// TIA Portal V20 export
FUNCTION_BLOCK "SysLinMotC1150"   // FB2080, FBD
TITLE = manage the positioning over the "extended bus positioning" [6Word]
{ S7_Optimized_Access := 'TRUE' }
AUTHOR : MiCROTEC
VERSION : 1.6
// -2019.12 : Martin
// stored: AutoNumber false, MemoryReserve 100, SetENOAutomatically false
   VAR_INPUT
      adr { ExternalAccessible := 'False'; ExternalVisible := 'False'; ExternalWritable := 'False'} : HW_IO;   // I/O address
      adrMc1 { ExternalAccessible := 'False'; ExternalVisible := 'False'; ExternalWritable := 'False'} : HW_IO;   // I/O address monitoring channel 1
      adrMc2 { ExternalAccessible := 'False'; ExternalVisible := 'False'; ExternalWritable := 'False'} : HW_IO;   // I/O address monitoring channel 2
      area { ExternalAccessible := 'False'; ExternalVisible := 'False'; ExternalWritable := 'False'} : Bool;   // 1=Safety area on
      areaDel { ExternalAccessible := 'False'; ExternalVisible := 'False'; ExternalWritable := 'False'} : Bool;   // 1=safety area on off-delayed
      auto { ExternalAccessible := 'False'; ExternalVisible := 'False'; ExternalWritable := 'False'} : Bool;   // automatic
      manP { ExternalAccessible := 'False'; ExternalVisible := 'False'; ExternalWritable := 'False'} : Bool;   // manual plus
      manM { ExternalAccessible := 'False'; ExternalVisible := 'False'; ExternalWritable := 'False'} : Bool;   // manual minus
      enable { ExternalAccessible := 'False'; ExternalVisible := 'False'; ExternalWritable := 'False'} : Bool;   // enable positioning
      enableP { ExternalAccessible := 'False'; ExternalVisible := 'False'; ExternalWritable := 'False'} : Bool;   // release plus
      enableM { ExternalAccessible := 'False'; ExternalVisible := 'False'; ExternalWritable := 'False'} : Bool;   // release minus
      ref { ExternalAccessible := 'False'; ExternalVisible := 'False'; ExternalWritable := 'False'} : Bool;   // reference
      ack { ExternalAccessible := 'False'; ExternalVisible := 'False'; ExternalWritable := 'False'} : Bool;   // fault acknowledge
      lampTest { ExternalAccessible := 'False'; ExternalVisible := 'False'; ExternalWritable := 'False'} : Bool;   // lamptest
      PwrSupMot { ExternalAccessible := 'False'; ExternalVisible := 'False'; ExternalWritable := 'False'} : Bool;   // 1=power supply motor ok / 1=motor protection switch ok
      PwrSupCtrl { ExternalAccessible := 'False'; ExternalVisible := 'False'; ExternalWritable := 'False'} : Bool;   // 1=power supply controller ok / 1=Motor protection switch brake ok
      tolerance { ExternalAccessible := 'False'; ExternalVisible := 'False'; ExternalWritable := 'False'} : Real;   // tolerance for output signal position ok
      mode { ExternalAccessible := 'False'; ExternalVisible := 'False'; ExternalWritable := 'False'} : Int;   // 1=VAI / 2=SIN VA / 3=Bestehorn VAJ
      target { ExternalAccessible := 'False'; ExternalVisible := 'False'; ExternalWritable := 'False'} : Real;   // target position [mm] / target position
      speed { ExternalAccessible := 'False'; ExternalVisible := 'False'; ExternalWritable := 'False'} : Real;   // target speed [m/s ] / target speed [ 1/min ]
      Acc { ExternalAccessible := 'False'; ExternalVisible := 'False'; ExternalWritable := 'False'} : Real;   // acceleration [m/s2] / start ramp [ms]
      Dec { ExternalAccessible := 'False'; ExternalVisible := 'False'; ExternalWritable := 'False'} : Real;   // deceleration [m/s2] / stop ramp [ms]
      jerk { ExternalAccessible := 'False'; ExternalVisible := 'False'; ExternalWritable := 'False'} : Real;   // jerk [m/s3]
   END_VAR
   VAR_OUTPUT
      comOk { ExternalAccessible := 'False'; ExternalVisible := 'False'; ExternalWritable := 'False'} : Bool;   // frequency converter communication ok
      ready { ExternalAccessible := 'False'; ExternalVisible := 'False'; ExternalWritable := 'False'} : Bool;   // frequency converter ready
      encAct { ExternalAccessible := 'False'; ExternalVisible := 'False'; ExternalWritable := 'False'} : DInt;   // actual position [inc]
      actual { ExternalAccessible := 'False'; ExternalVisible := 'False'; ExternalWritable := 'False'} : Real;   // actual position
      refOk { ExternalAccessible := 'False'; ExternalVisible := 'False'; ExternalWritable := 'False'} : Bool;   // reference ok
      refRun { ExternalAccessible := 'False'; ExternalVisible := 'False'; ExternalWritable := 'False'} : Bool;   // reference run active
      posOk { ExternalAccessible := 'False'; ExternalVisible := 'False'; ExternalWritable := 'False'} : Bool;   // position ok
      lamp { ExternalAccessible := 'False'; ExternalVisible := 'False'; ExternalWritable := 'False'} : Bool;   // indication lamp
      err { ExternalAccessible := 'False'; ExternalVisible := 'False'; ExternalWritable := 'False'} : Bool;   // fault
      errEnc { ExternalAccessible := 'False'; ExternalVisible := 'False'; ExternalWritable := 'False'} : Bool;   // fault encoder
      war { ExternalAccessible := 'False'; ExternalVisible := 'False'; ExternalWritable := 'False'} : Bool;   // warning
   END_VAR
   VAR_IN_OUT
      Mot : "TypeMotor";   // data motor
   END_VAR
   VAR
      var { ExternalAccessible := 'False'; ExternalVisible := 'False'; ExternalWritable := 'False'} : Struct
         "bool" : Bool;
         "byte" : Byte;
         "word" : Word;
         "dword" : DWord;
         "int" : Int;
         "dint" : DInt;
         "real" : Real;
         s5time : S5Time;
         "time" : Time;
         hm : Array[1..16] of Bool;
         fm : Array[1..16] of Bool;
      END_STRUCT;
      Rd { ExternalAccessible := 'False'; ExternalVisible := 'False'; ExternalWritable := 'False'} : "TypeLinmotRd";
      RdMc1 { ExternalAccessible := 'False'; ExternalVisible := 'False'; ExternalWritable := 'False'} : DInt;   // actual velocity
      RdMc2 { ExternalAccessible := 'False'; ExternalVisible := 'False'; ExternalWritable := 'False'} : DInt;   // actual error code
      Sd { ExternalAccessible := 'False'; ExternalVisible := 'False'; ExternalWritable := 'False'} : "TypeLinmotSd";
      T { ExternalAccessible := 'False'; ExternalVisible := 'False'; ExternalWritable := 'False'} : Array[1..8] of IEC_TIMER;
      errNrOld { ExternalAccessible := 'False'; ExternalVisible := 'False'; ExternalWritable := 'False'} : UDInt;
      man { ExternalAccessible := 'False'; ExternalVisible := 'False'; ExternalWritable := 'False'} : Bool;
      autoOld { ExternalAccessible := 'False'; ExternalVisible := 'False'; ExternalWritable := 'False'} : Bool;
      errGen { ExternalAccessible := 'False'; ExternalVisible := 'False'; ExternalWritable := 'False'} : Bool;
      enOnDel { ExternalAccessible := 'False'; ExternalVisible := 'False'; ExternalWritable := 'False'} : Bool;
      MotEnable { ExternalAccessible := 'False'; ExternalVisible := 'False'; ExternalWritable := 'False'} : Bool;
      MotSwitchOn { ExternalAccessible := 'False'; ExternalVisible := 'False'; ExternalWritable := 'False'} : Bool;
      statReady { ExternalAccessible := 'False'; ExternalVisible := 'False'; ExternalWritable := 'False'} : Bool;
      statCtrlAuto { ExternalAccessible := 'False'; ExternalVisible := 'False'; ExternalWritable := 'False'} : Bool;
      TarPos { ExternalAccessible := 'False'; ExternalVisible := 'False'; ExternalWritable := 'False'} : Real;
      TarCurrent { ExternalAccessible := 'False'; ExternalVisible := 'False'; ExternalWritable := 'False'} : Real;
      TimeResetHome { ExternalAccessible := 'False'; ExternalVisible := 'False'; ExternalWritable := 'False'} : TON_TIME;
      targetOld { ExternalAccessible := 'False'; ExternalVisible := 'False'; ExternalWritable := 'False'} : Real;
      StartPos { ExternalAccessible := 'False'; ExternalVisible := 'False'; ExternalWritable := 'False'} : Bool;
      PosTolOk { ExternalAccessible := 'False'; ExternalVisible := 'False'; ExternalWritable := 'False'} : Bool;
      TimeStartPos { ExternalAccessible := 'False'; ExternalVisible := 'False'; ExternalWritable := 'False'} : TP_TIME;
      McPar4 { ExternalAccessible := 'False'; ExternalVisible := 'False'; ExternalWritable := 'False'} : Real;
      Mc1 { ExternalAccessible := 'False'; ExternalVisible := 'False'; ExternalWritable := 'False'} : DInt;
      Mc2 { ExternalAccessible := 'False'; ExternalVisible := 'False'; ExternalWritable := 'False'} : DInt;
   END_VAR
   VAR_TEMP
      tempSdRetVal : Int;
      tempRdRetVal1 : Int;
      tempRdRetVal2 : Int;
      tempRdRetVal3 : Int;
      tempName : WString[20];
      tempDescription : WString[60];
      label : WString[26];
      tempString : WString;
      tempStrgPointer : Int;
      tempAck : Bool;
      tempStat : Bool;
      tempWar : Bool;
      tempOp : DInt;
      tempRd : Array[0..3] of Byte;
      tempDint : DInt;
      tempSd : Array[0..3] of Byte;
   END_VAR
   VAR_TEMP   // added for the SCL form of the ladder/FBD networks
      _w1 : Bool;
      _w2 : Bool;
   END_VAR
BEGIN

REGION Network 1 (SCL): description
   // Linmot  PL01-20x800/740-HP  Motor Stange Noale
   // control of a linmot motor
   // controller:  Linmot C1150-PN-XC-1S
   // stator:      Linmot PS01-37Sx120F-HP-N-AGI
   // stroke:      Linmot PL01-20x360/300-HP
   // creator:     Alexander Kiebacher
   // version:     1.0
   //
END_REGION

REGION Network 2: exit
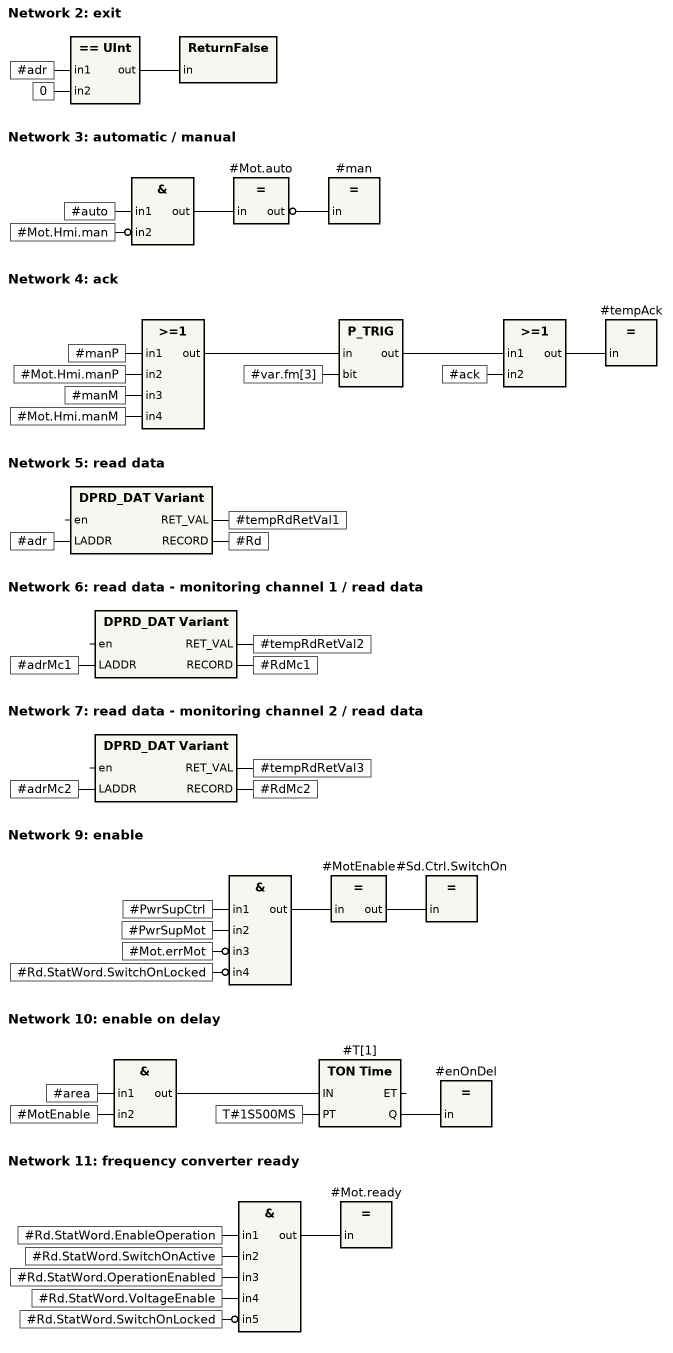
   IF #adr = 0 THEN
       ENO := FALSE;
       RETURN;
   END_IF;
END_REGION

REGION Network 3: automatic / manual
   #_w1 := #auto AND NOT #Mot.Hmi.man;
   #Mot.auto := #_w1;
   #man := NOT #_w1;
END_REGION

REGION Network 4: ack
   #_w1 := #manP OR #Mot.Hmi.manP OR #manM OR #Mot.Hmi.manM;
   #_w2 := #_w1 AND NOT #var.fm[3];   // rising edge
   #var.fm[3] := #_w1;
   #tempAck := #_w2 OR #ack;
END_REGION

REGION Network 5: read data
   #tempRdRetVal1 := DPRD_DAT(LADDR := #adr, RECORD => #Rd);
END_REGION

REGION Network 6: read data - monitoring channel 1 / read data
   #tempRdRetVal2 := DPRD_DAT(LADDR := #adrMc1, RECORD => #RdMc1);
END_REGION

REGION Network 7: read data - monitoring channel 2 / read data
   #tempRdRetVal3 := DPRD_DAT(LADDR := #adrMc2, RECORD => #RdMc2);
END_REGION

REGION Network 8 (SCL): read

   // actual position
   #tempRd[0] := #Rd.Actpos.%B0;
   #tempRd[1] := #Rd.Actpos.%B1;
   #tempRd[2] := #Rd.Actpos.%B2;
   #tempRd[3] := #Rd.Actpos.%B3;

   #Rd.Actpos.%B0 := #tempRd[3];
   #Rd.Actpos.%B1 := #tempRd[2];
   #Rd.Actpos.%B2 := #tempRd[1];
   #Rd.Actpos.%B3 := #tempRd[0];

   #encAct := #Rd.Actpos;
   #actual := DINT_TO_REAL(#Rd.Actpos) / 10000.0;

   // target position
   #tempRd[0] := #Rd.Tarpos.%B0;
   #tempRd[1] := #Rd.Tarpos.%B1;
   #tempRd[2] := #Rd.Tarpos.%B2;
   #tempRd[3] := #Rd.Tarpos.%B3;

   #Rd.Tarpos.%B0 := #tempRd[3];
   #Rd.Tarpos.%B1 := #tempRd[2];
   #Rd.Tarpos.%B2 := #tempRd[1];
   #Rd.Tarpos.%B3 := #tempRd[0];

   #TarPos := DINT_TO_REAL(#Rd.Tarpos) / 10000.0;

   // target current
   #tempRd[0] := #Rd.TarCurrent.%B0;
   #tempRd[1] := #Rd.TarCurrent.%B1;
   #tempRd[2] := #Rd.TarCurrent.%B2;
   #tempRd[3] := #Rd.TarCurrent.%B3;

   #Rd.TarCurrent.%B0 := #tempRd[3];
   #Rd.TarCurrent.%B1 := #tempRd[2];
   #Rd.TarCurrent.%B2 := #tempRd[1];
   #Rd.TarCurrent.%B3 := #tempRd[0];

   #TarCurrent := DINT_TO_REAL(#Rd.TarCurrent) / 1000.0;

   // monitoring channel 1 - target velocity [1000*m/s]
   #tempRd[0] := #RdMc1.%B0;
   #tempRd[1] := #RdMc1.%B1;
   #tempRd[2] := #RdMc1.%B2;
   #tempRd[3] := #RdMc1.%B3;

   #RdMc1.%B0 := #tempRd[3];
   #RdMc1.%B1 := #tempRd[2];
   #RdMc1.%B2 := #tempRd[1];
   #RdMc1.%B3 := #tempRd[0];

   #Mc1 := #RdMc1;

   IF #Rd.StatWord.MotionActive THEN
       IF #Mc1 >= 100 THEN
           #Mot.speedAct := DINT_TO_INT(#Mc1/1000);
       ELSIF #Mc1 <= -100 THEN
           #Mot.speedAct := DINT_TO_INT(#Mc1/1000);
       END_IF;
   ELSE
       #Mot.speedAct := 0;
   END_IF;

   // monitoring channel 2 - actual error code
   #tempRd[0] := #RdMc2.%B0;
   #tempRd[1] := #RdMc2.%B1;
   #tempRd[2] := #RdMc2.%B2;
   #tempRd[3] := #RdMc2.%B3;

   #RdMc2.%B0 := #tempRd[3];
   #RdMc2.%B1 := #tempRd[2];
   #RdMc2.%B2 := #tempRd[1];
   #RdMc2.%B3 := #tempRd[0];

   #Mc2 := #RdMc2;
END_REGION

REGION Network 9: enable
   #MotEnable := #PwrSupCtrl AND #PwrSupMot AND NOT #Mot.errMot AND NOT #Rd.StatWord.SwitchOnLocked;
   #Sd.Ctrl.SwitchOn := #MotEnable;
END_REGION

REGION Network 10: enable on delay
   #T[1].TON(IN := #area AND #MotEnable, PT := T#1S500MS);
   #enOnDel := #T[1].Q;
END_REGION

REGION Network 11: frequency converter ready
   #Mot.ready := #Rd.StatWord.EnableOperation AND #Rd.StatWord.SwitchOnActive AND #Rd.StatWord.OperationEnabled AND #Rd.StatWord.VoltageEnable AND NOT #Rd.StatWord.SwitchOnLocked;
END_REGION

REGION Network 12: ready
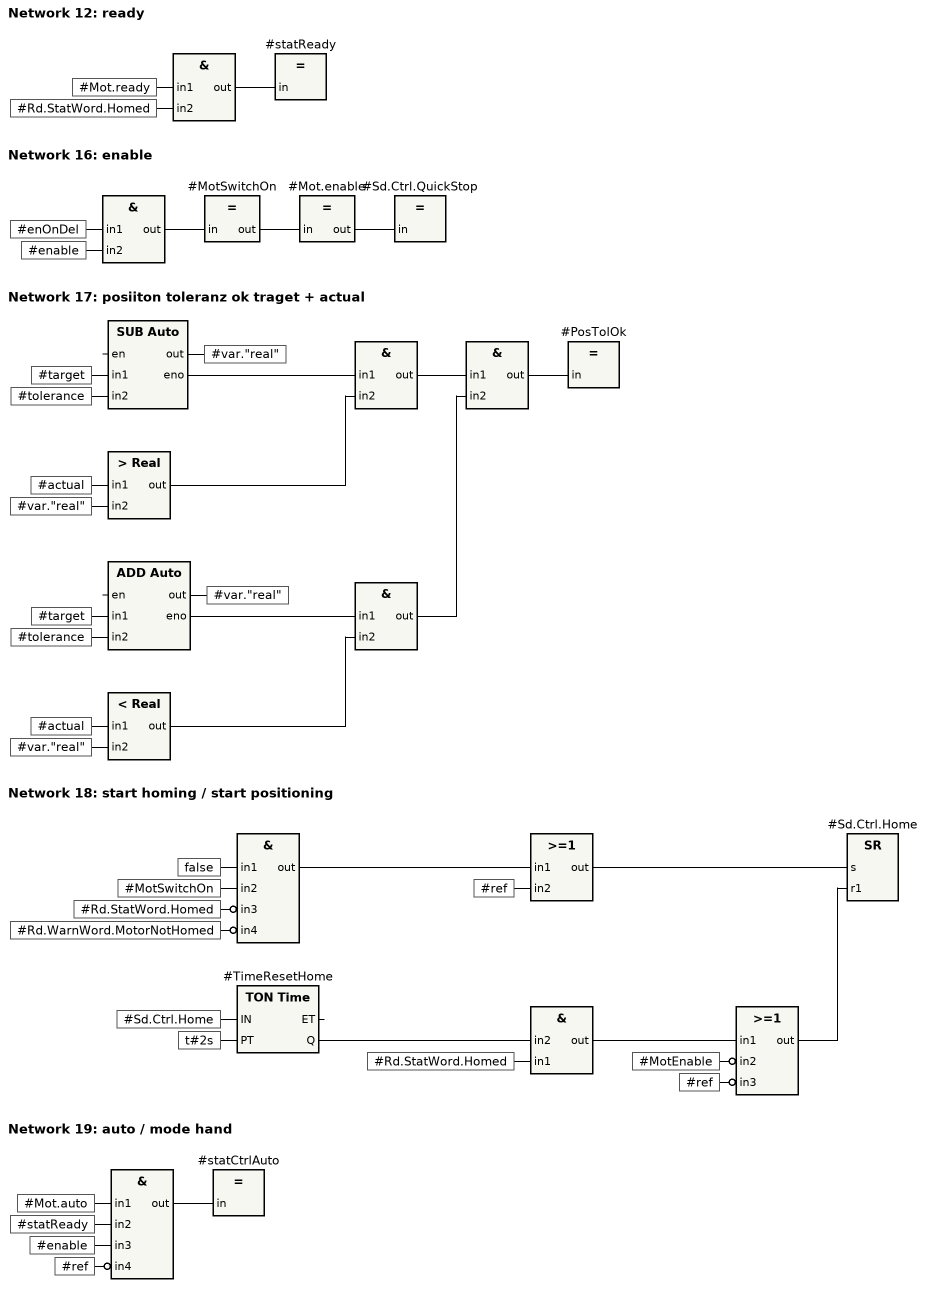
   #statReady := #Mot.ready AND #Rd.StatWord.Homed;
END_REGION

NETWORK
TITLE = test status var

      L     #Rd.StatVar.MainState;  // Op. Main State
      L     #Rd.StatVar.SubState;  // Op. Sub State

      T     #tempOp;


NETWORK
TITLE = test status word

// not used
      O     #Rd.StatWord.EventHandlerActive;
      O     #Rd.StatWord.SpecialMotionActive;
      O     #Rd.StatWord.MotionActive;
      O     #Rd.StatWord.RangeIndicator1;
      O     #Rd.StatWord.RangeIndicator2;
      =     #tempStat;


NETWORK
TITLE = test warning word

// not used
      O     #Rd.StatWord.Warning;
      O     #Rd.WarnWord.MotorHotSensor;
      O     #Rd.WarnWord.MotorShortTimerOverload;
      O     #Rd.WarnWord.MotorSupplyVoltageLow;
      O     #Rd.WarnWord.MotorSupplyVoltageHigh;
      O     #Rd.WarnWord.PositionLagAlways;
      O     #Rd.WarnWord.Res5;
      O     #Rd.WarnWord.DriveHot;
      O     #Rd.WarnWord.PTC_Sensor1Hot;
      O     #Rd.WarnWord.PTC_Sensor2Hot;
      O     #Rd.WarnWord.Res10;
      O     #Rd.WarnWord.Res11;
      O     #Rd.WarnWord.Res12;
      O     #Rd.WarnWord.Res13;
      O     #Rd.WarnWord.InterfaceWarnFlag;
      O     #Rd.WarnWord.ApplicationWarnFlag;
      =     #tempWar;


REGION Network 16: enable
   #MotSwitchOn := #enOnDel AND #enable;
   #Mot.enable := #MotSwitchOn;
   #Sd.Ctrl.QuickStop := #MotSwitchOn;
END_REGION

REGION Network 17: posiiton toleranz ok traget + actual
   #var."real" := #target - #tolerance;
   #_w1 := #actual > #var."real";
   #var."real" := #target + #tolerance;
   #PosTolOk := #_w1 AND (#actual < #var."real");
END_REGION

REGION Network 18: start homing / start positioning
   // auto reference?
   #TimeResetHome(IN := #Sd.Ctrl.Home, PT := t#2s);   // TON
   IF (false AND #MotSwitchOn AND NOT #Rd.StatWord.Homed AND NOT #Rd.WarnWord.MotorNotHomed) OR #ref THEN
       #Sd.Ctrl.Home := TRUE;   // SR flip-flop
   END_IF;
   IF (#TimeResetHome.Q AND #Rd.StatWord.Homed) OR NOT #MotEnable OR NOT #ref THEN
       #Sd.Ctrl.Home := FALSE;
   END_IF;
END_REGION

REGION Network 19: auto / mode hand
   #statCtrlAuto := #Mot.auto AND #statReady AND #enable AND NOT #ref;
END_REGION

REGION Network 20: start positioning
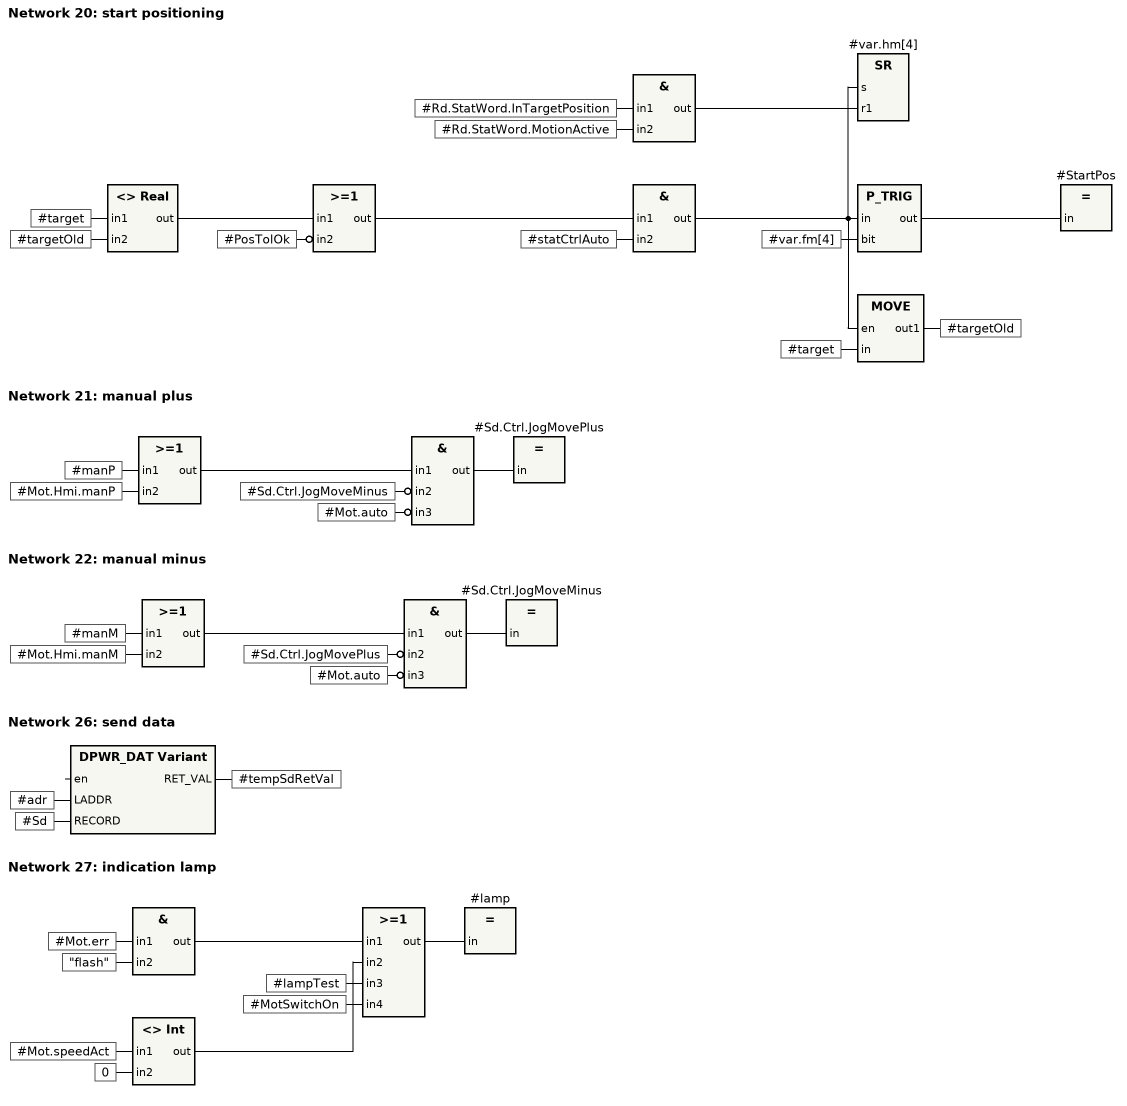
   #_w1 := ((#target <> #targetOld) OR NOT #PosTolOk) AND #statCtrlAuto;
   IF #_w1 THEN
       #var.hm[4] := TRUE;   // SR flip-flop
   END_IF;
   IF #Rd.StatWord.InTargetPosition AND #Rd.StatWord.MotionActive THEN #var.hm[4] := FALSE; END_IF;
   #_w2 := #_w1 AND NOT #var.fm[4];   // rising edge
   #var.fm[4] := #_w1;
   #StartPos := #_w2;
   IF #_w1 THEN #targetOld := #target; END_IF;
END_REGION

REGION Network 21: manual plus
   #Sd.Ctrl.JogMovePlus := (#manP OR #Mot.Hmi.manP) AND NOT #Sd.Ctrl.JogMoveMinus AND NOT #Mot.auto;
END_REGION

REGION Network 22: manual minus
   #Sd.Ctrl.JogMoveMinus := (#manM OR #Mot.Hmi.manM) AND NOT #Sd.Ctrl.JogMovePlus AND NOT #Mot.auto;
END_REGION

REGION Network 23 (SCL)

   #Sd.Ctrl.EnableOperation := TRUE;          // Forced
   #Sd.Ctrl.Abort := TRUE;                    // Forced
   #Sd.Ctrl.Freeze := TRUE;                   // Forced

   // not used
   #Sd.Ctrl.VoltageEnable := FALSE;            // STO
   #Sd.Ctrl.GoToPosition := FALSE;
   #Sd.Ctrl.SpecialMove := FALSE;
   #Sd.Ctrl.ClearanceCheck := FALSE;
   #Sd.Ctrl.GoToInitialPosition := FALSE;
   #Sd.Ctrl.Linearizing := FALSE;
   #Sd.Ctrl.PhaseSearch := FALSE;
END_REGION

REGION Network 24 (SCL): write - MC Header / write

   // Command Count
   // A new command will only be executed, if the value of the command count has changed. In the easiest way bit 0 can be toggled
   #Sd.McHd.CC0 := #StartPos;
   #Sd.McHd.CC1 := FALSE;
   #Sd.McHd.CC2 := FALSE;
   #Sd.McHd.CC3 := FALSE;

   // Master ID
   #Sd.McHd.MasterID := B#16#00;
   IF #mode = 1 THEN
       // VAI
       #Sd.McHd.MasterID := B#16#01;
   ELSIF #mode = 2 THEN
       // SIN VA
       #Sd.McHd.MasterID := B#16#0E;
   ELSIF #mode = 3 THEN
       // Bestehorn VAJ
       #Sd.McHd.MasterID := B#16#0F;
   END_IF;

   // not used Sub ID
   #Sd.McHd.SubID0 := FALSE;
   #Sd.McHd.SubID1 := FALSE;
   #Sd.McHd.SubID2 := FALSE;
   #Sd.McHd.SubID3 := FALSE;
END_REGION

REGION Network 25 (SCL): write - MC Parameter / write

   #Sd.McPar1 := L#0;
   #Sd.McPar2 := L#0;
   #Sd.McPar3 := L#0;
   #Sd.McPar4 := L#0;

   // McPar1 - target
   // 
   #tempDint := REAL_TO_DINT(#target * 10000.0);
   #tempSd[0] := #tempDint.%B0;
   #tempSd[1] := #tempDint.%B1;
   #tempSd[2] := #tempDint.%B2;
   #tempSd[3] := #tempDint.%B3;

   #Sd.McPar1.%B0 := #tempSd[3];
   #Sd.McPar1.%B1 := #tempSd[2];
   #Sd.McPar1.%B2 := #tempSd[1];
   #Sd.McPar1.%B3 := #tempSd[0];

   // McPar2 - speed
   // 
   #tempDint := REAL_TO_DINT(#speed * 1000000.0);
   #tempSd[0] := #tempDint.%B0;
   #tempSd[1] := #tempDint.%B1;
   #tempSd[2] := #tempDint.%B2;
   #tempSd[3] := #tempDint.%B3;

   #Sd.McPar2.%B0 := #tempSd[3];
   #Sd.McPar2.%B1 := #tempSd[2];
   #Sd.McPar2.%B2 := #tempSd[1];
   #Sd.McPar2.%B3 := #tempSd[0];

   // McPar3
   // VAI              - acc
   // SIN VA           - acc/dec
   // Bestehorn VAJ    - acc/dec
   #tempDint := REAL_TO_DINT(#Acc * 100000.0);
   #tempSd[0] := #tempDint.%B0;
   #tempSd[1] := #tempDint.%B1;
   #tempSd[2] := #tempDint.%B2;
   #tempSd[3] := #tempDint.%B3;

   #Sd.McPar3.%B0 := #tempSd[3];
   #Sd.McPar3.%B1 := #tempSd[2];
   #Sd.McPar3.%B2 := #tempSd[1];
   #Sd.McPar3.%B3 := #tempSd[0];

   // McPar4
   #McPar4 := 0.0;
   #tempDint := 0;
   IF #mode = 1 THEN
       // VAI
       #McPar4 := #Dec;
       #tempDint := REAL_TO_DINT(#McPar4 * 100000.0);
   ELSIF #mode = 2 THEN
       // SIN VA
       #McPar4 := 0.0;
       #tempDint := REAL_TO_DINT(#McPar4 * 100000.0);
   ELSIF #mode = 3 THEN
       // Bestehorn VAJ
       #McPar4 := #jerk;
       #tempDint := REAL_TO_DINT(#McPar4 * 10000.0);
   END_IF;

   #tempSd[0] := #tempDint.%B0;
   #tempSd[1] := #tempDint.%B1;
   #tempSd[2] := #tempDint.%B2;
   #tempSd[3] := #tempDint.%B3;

   #Sd.McPar4.%B0 := #tempSd[3];
   #Sd.McPar4.%B1 := #tempSd[2];
   #Sd.McPar4.%B2 := #tempSd[1];
   #Sd.McPar4.%B3 := #tempSd[0];
END_REGION

REGION Network 26: send data
   #tempSdRetVal := DPWR_DAT(LADDR := #adr, RECORD := #Sd);
END_REGION

REGION Network 27: indication lamp
   #lamp := (#Mot.err AND "flash") OR (#Mot.speedAct <> 0) OR #lampTest OR #MotSwitchOn;
END_REGION

REGION Network 28: communication ok
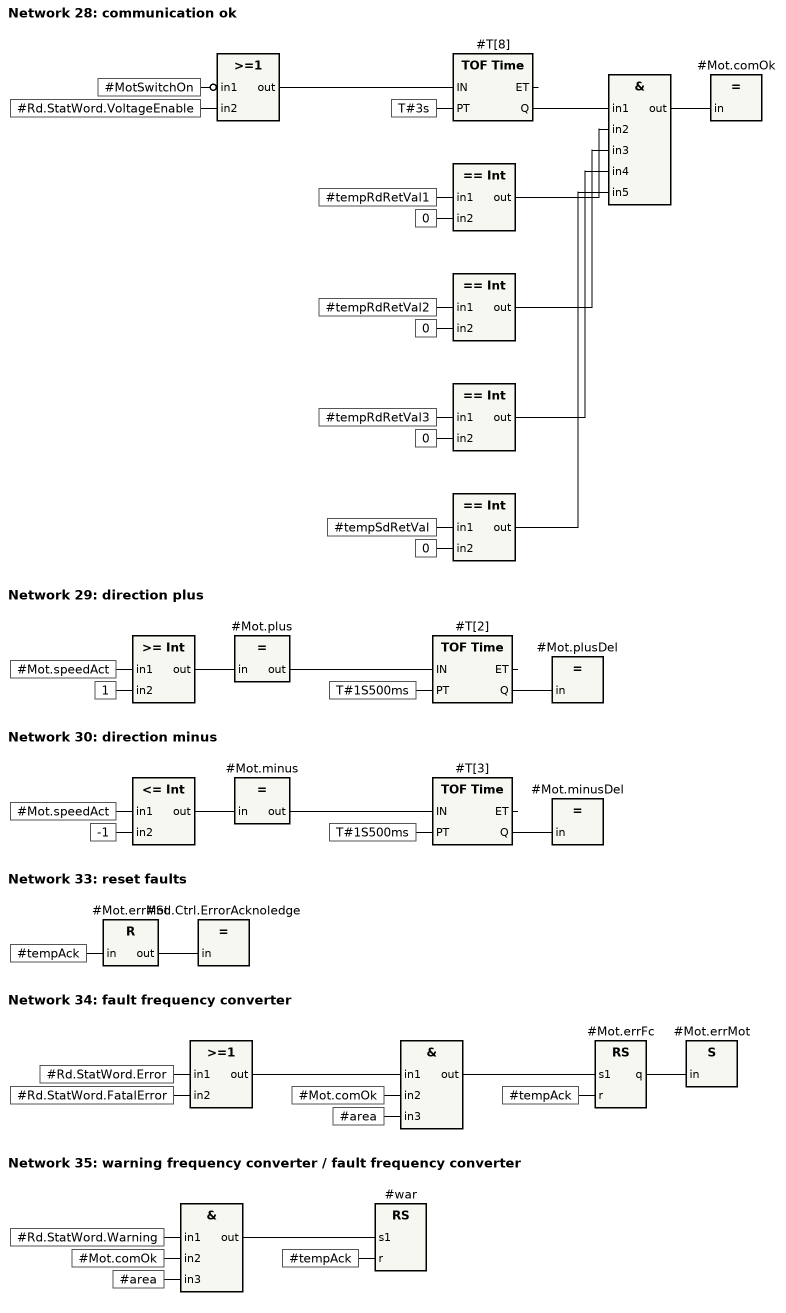
   #T[8].TOF(IN := NOT #MotSwitchOn OR #Rd.StatWord.VoltageEnable, PT := T#3s);
   #Mot.comOk := #T[8].Q AND (#tempRdRetVal1 = 0) AND (#tempRdRetVal2 = 0) AND (#tempRdRetVal3 = 0) AND (#tempSdRetVal = 0);
END_REGION

REGION Network 29: direction plus
   #Mot.plus := #Mot.speedAct >= 1;
   #T[2].TOF(IN := #Mot.plus, PT := T#1S500ms);
   #Mot.plusDel := #T[2].Q;
END_REGION

REGION Network 30: direction minus
   #Mot.minus := #Mot.speedAct <= (-1);
   #T[3].TOF(IN := #Mot.minus, PT := T#1S500ms);
   #Mot.minusDel := #T[3].Q;
END_REGION

REGION Network 32: --faults--
END_REGION

REGION Network 33: reset faults
   IF #tempAck THEN #Mot.errMot := FALSE; END_IF;
   #Sd.Ctrl.ErrorAcknoledge := #tempAck;
END_REGION

REGION Network 34: fault frequency converter
   IF #tempAck THEN
       #Mot.errFc := FALSE;   // RS flip-flop
   END_IF;
   IF (#Rd.StatWord.Error OR #Rd.StatWord.FatalError) AND #Mot.comOk AND #area THEN
       #Mot.errFc := TRUE;
   END_IF;
   IF #Mot.errFc THEN #Mot.errMot := TRUE; END_IF;
END_REGION

REGION Network 35: warning frequency converter / fault frequency converter
   IF #tempAck THEN
       #war := FALSE;   // RS flip-flop
   END_IF;
   IF #Rd.StatWord.Warning AND #Mot.comOk AND #area THEN #war := TRUE; END_IF;
END_REGION

REGION Network 36: fault motor protection motor
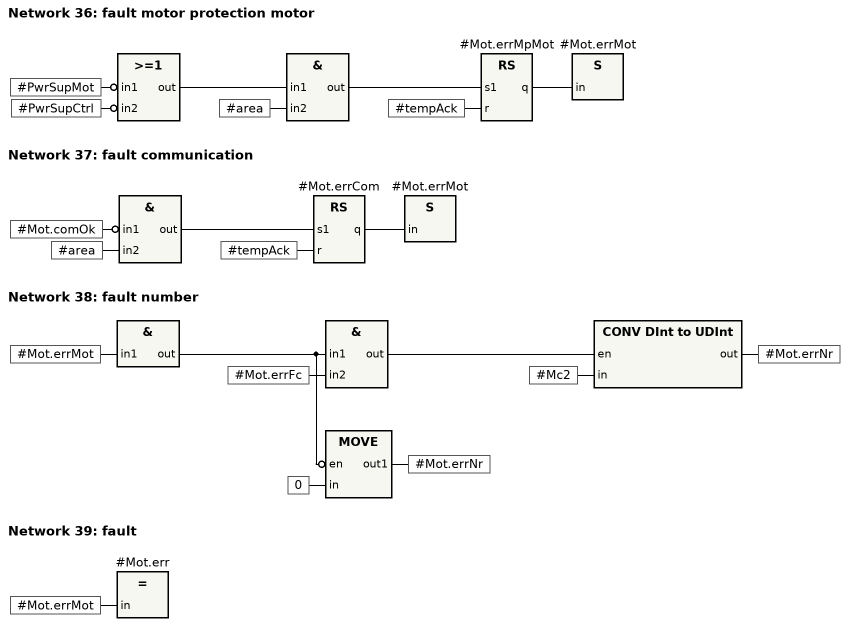
   IF #tempAck THEN
       #Mot.errMpMot := FALSE;   // RS flip-flop
   END_IF;
   IF (NOT #PwrSupMot OR NOT #PwrSupCtrl) AND #area THEN #Mot.errMpMot := TRUE; END_IF;
   IF #Mot.errMpMot THEN #Mot.errMot := TRUE; END_IF;
END_REGION

REGION Network 37: fault communication
   IF #tempAck THEN
       #Mot.errCom := FALSE;   // RS flip-flop
   END_IF;
   IF NOT #Mot.comOk AND #area THEN #Mot.errCom := TRUE; END_IF;
   IF #Mot.errCom THEN #Mot.errMot := TRUE; END_IF;
END_REGION

REGION Network 38: fault number
   IF #Mot.errMot AND #Mot.errFc THEN #Mot.errNr := DINT_TO_UDINT(#Mc2); END_IF;
   IF NOT #Mot.errMot THEN #Mot.errNr := 0; END_IF;
END_REGION

REGION Network 39: fault
   #Mot.err := #Mot.errMot;
END_REGION

REGION Network 40 (SCL): write outputs
   #comOk := #Mot.comOk;
   #ready := #Mot.ready;
   #err := #Mot.err;
   #errEnc := #Mot.err;
   #refOk := #Rd.StatWord.Homed;
   #refRun := #Sd.Ctrl.Home;
   #posOk := (#Rd.StatWord.InTargetPosition OR TRUE) AND #PosTolOk;
END_REGION

REGION Network 41 (SCL): in/out data
   #Mot.run := #Mot.plus OR #Mot.minus;
   #Mot.runDel := #Mot.plusDel OR #Mot.minusDel;
   #Mot.enStartP := false;
   #Mot.enStartM := false;
   #Mot.speedTar := DINT_TO_INT(#speed);
   #Mot.area := #area;

   IF #auto AND NOT #autoOld THEN
       #Mot.Hmi.man := false;
       #Mot.Hmi.manP := false;
       #Mot.Hmi.manM := false;
   END_IF;
   #autoOld := #auto;
END_REGION
END_FUNCTION_BLOCK
